ABB RAPID module: Wobj_wobj_A.mod

MODULE Wobj_wobj_A
	! Points are read in order of declaration.
  ! Please do not change the order of points!

  LOCAL PERS robtarget pWobj_U_PointX1:=[[1393.435,-1975.626,-698.8897],[0.000257953244727105,-0.72753918170929,0.686065554618835,0.000876909703947604],[-1,0,2,0],[0,9E+09,9E+09,9E+09,9E+09,9E+09]];
	LOCAL PERS robtarget pWobj_U_PointX2:=[[1557.349,-1975.654,-698.8638],[0.000256044848356396,-0.727539122104645,0.68606561422348,0.000866393325850368],[-1,0,2,0],[0,9E+09,9E+09,9E+09,9E+09,9E+09]];
	LOCAL PERS robtarget pWobj_U_PointY1:=[[1557.375,-1754.001,-698.8805],[0.00025822312454693,-0.727548539638519,0.686055660247803,0.000876544858328998],[-1,0,2,0],[0,9E+09,9E+09,9E+09,9E+09,9E+09]];

ENDMODULE
